// Block: Area02_HU_PERS

DATA_BLOCK Area02_HU_PERS
VERSION : 0.1
   NON_RETAIN
   VAR
      PersistentValues : Struct
         Par_Pump : HU_Pump_Par;
         Par_Tank : HU_Tank_Par;
      END_STRUCT;
      HMI : Struct
         ActuaPressure : Real;
      END_STRUCT;
   END_VAR

BEGIN
   // No initialization required
END_DATA_BLOCK
